// TwinCAT 3 PLC project DiagnosisTools
// Title: TwinCATDiagnosisTools
// Company: Beckhoff Automation K.K.
// Author: Takashi Ichihashi
// ProjectVersion: 1.0.0.1
// ProgramVersion: 3.1.4024.0
// libraries:
//   Tc2_EtherCAT, * (Beckhoff Automation GmbH)
//   Tc2_Standard, * (Beckhoff Automation GmbH)
//   Tc2_System, * (Beckhoff Automation GmbH)
//   Tc2_Utilities, * (Beckhoff Automation GmbH)
//   Tc3_Module, * (Beckhoff Automation GmbH)
// project tree:
//   DUTs/ CoeSdoCommand.TcDUT, sdo_EL6695_diag.TcDUT, sdo_slave_identity.TcDUT, sdo_xplanar_aps_diag.TcDUT
//   GVLs/ ParameterList.TcGVL
//   / PlcTask.TcTTO
//   POUs/ FB_CoeSdoAccess.TcPOU, FB_mqtt_publish.TcPOU, FB_serializer.TcPOU (not stored), ITF_CoeSdoEventHandler.TcIO, queue.TcPOU, MAIN.TcPOU, sdo_watch_time_logging.TcPOU
// real-time tasks:
//   TASK PlcTask: cycle T#10ms, priority 20, ADS port 350
// I/O:
//   DEVICE Device 3 (EtherCAT), AmsNetId 10.200.64.8.4.1
//     Term 1 (EK1100) [EK1100 EtherCAT Coupler (2A E-Bus)]
//       Term 2 (EL2521) [EL2521 1Ch. Pulse Train Output]
//       Term 3 (EL4122) [EL4122 2Ch. Ana. Output  4-20mA, 16bit]
//       Term 4 (EL9576) [EL9576 Brake chopper terminal]
//       Term 5 (EL3152) [EL3152 2Ch. Ana Input 4-20mA]
//       Term 6 (EL2004) [EL2004 4Ch. Dig. Output 24V, 0.5A]
//       Term 7 (EL5101) [EL5101 1Ch. Inc. Encoder 5V]
//       Term 8 (EL6695) [EL6695 EtherCAT Bridge terminal (Primary)]
//       Term 9 (EL9011) [EL9011 End Terminal]

CONFIGURATION DiagnosisTools
    RESOURCE PLC ON TwinCAT3
        TASK PlcTask(INTERVAL := T#10ms, PRIORITY := 20);
        PROGRAM MAIN WITH PlcTask : MAIN;
    END_RESOURCE
END_CONFIGURATION

// ---- DUTs/CoeSdoCommand.TcDUT
(*
SdoRead/WriteRequest
*)
TYPE CoeSdoCommand:
STRUCT
	sNetId				: T_AmsNetId;	// AMS Net ID of EtherCAT Master
	nSlaveAddr			: UINT;			// EtherCAT sub device address
	bCompleteAccess		: BOOL;			// Enable complete access
	nSubIndex			: BYTE;			// Subindex of OD
	nIndex				: WORD;			// Index of OD
	pDstBuf				: PVOID;		// Pointer to data body 
	cbBufLen			: UDINT;		// Size of data body
	datetime			: TIMESTRUCT;	// to be recorded as received date time
	event_handler		: ITF_CoeSdoEventHandler; // Event handler interface
	bError				: BOOL;			// Made true if sdo communication error
	nErrId				: UDINT;		// Set error code if sdo communication error activated
END_STRUCT
END_TYPE

// ---- DUTs/sdo_EL6695_diag.TcDUT
{attribute 'pack_mode' := '2'}
TYPE sdo_EL6695_diag :
STRUCT
	identify : USINT;
	status : UINT;
	cpu_usage : UINT;
	heap_usage : UINT;
	aoe_packets: UINT;
	eoe_packets : UINT;
	foe_packets : UINT;
	soe_packets : UINT;
	voe_packets : UINT;
	other_pacekts: UINT;
	mbx_info : UINT;
	pd_copy_time_my: UINT;
	pd_copy_time_remote :UINT;
	info_2 : UINT;
	info_3 : UINT;
	info_4 : UINT;
	info_5 : UINT;
	info_6 : UINT;
	info_7 : UINT;
	info_8 : UINT;
	info_9 : UINT;
	info_10 : UINT;
	info_11 : UINT;
	info_12 : UINT;
	info_13 : UINT;
	info_14 : UINT;
	info_15 : UINT;
	info_16: UINT;
	info_17 : UINT;
	info_18 : UINT;
END_STRUCT
END_TYPE

// ---- DUTs/sdo_slave_identity.TcDUT
{attribute 'pack_mode' := '2'}
TYPE sdo_slave_identity :
STRUCT
	identify : USINT;
	vendor_id : UDINT;
	product_code : UDINT;
	revision : UDINT;
	serial_number : UDINT;
END_STRUCT
END_TYPE

// ---- DUTs/sdo_xplanar_aps_diag.TcDUT
{attribute 'pack_mode' := '2'}
TYPE sdo_xplanar_aps_diag :
STRUCT
  identity: USINT;
  dc_link_voltage: UDINT;
  power_supply_current: UDINT;
  temperature_north: UINT;
  temperature_east: UINT;
  temperature_south: UINT;
  temperature_west: UINT;
  temperature_center: UINT;
  temperature_power: UINT;
  fan_rpm: UINT;
  fan_duty_cycle: USINT;
  supply_voltage_us: UDINT;
  auxiliary_voltage: UDINT;
  acceleration_x: UDINT;
  acceleration_y: UDINT;
  acceleration_z: UDINT;
  time_to_shutdown: UDINT;
  fb_fw_rev: UDINT;
END_STRUCT
END_TYPE

// ---- GVLs/ParameterList.TcGVL
{attribute 'qualified_only'}
VAR_GLOBAL CONSTANT
	COMMAND_QUEUE_BUFFER_SIZE :UINT := 10;
	MAX_OBSERVATION_SDO :UINT := 100;
END_VAR

// ---- POUs/ITF_CoeSdoEventHandler.TcIO
INTERFACE ITF_CoeSdoEventHandler

METHOD sdo_data_received : BOOL
VAR_INPUT
	command : REFERENCE TO CoeSdoCommand;
END_VAR
END_METHOD

END_INTERFACE

// ---- POUs/MAIN.TcPOU
PROGRAM MAIN
VAR CONSTANT
	EC_MASTER_NETID : T_AmsNetId := '10.200.64.8.4.1';	
END_VAR
VAR

	// COE SDO communication controller object 
	sdo_controller : FB_CoeSdoAccess(sNetId := EC_MASTER_NETID); // EtherCAT Master Object for SDO control


	(* 
		For initialization process( Get all subdevices identity from SDO )
	*)

	bInitialize :BOOL := TRUE;
	s_adr :UINT;

	// define data store.
	sdo_slave_id_data : ARRAY [1002..1008] OF sdo_slave_identity;

	
	
	(*
		 Observation by EL6695 diagnosis data
	*)
	
	// define data store.
	sdo_EL6695_diag_data : sdo_EL6695_diag;
	
	// define event handler when sdo data received by "ITF_CoeSdoEventHandler" implementation.  
	sdo_protocol_with_time_detection: sdo_watch_time_logging;

	// cycle timer for "sdo_EL6695_diag_data" reading.
	read_cycle_timer : TON;
	
	// get ISO 8601 format datetime and cycle time for sdo data received generated by "sdo_protocol_with_time_detection.sdo_data_received()" method.
	datetime_string: STRING(39);
	cycle_time :ULINT;
	
END_VAR

sdo_controller();

// Get Identity data for all sub devices
IF bInitialize THEN
	FOR s_adr := 1002 TO 1008 DO
		sdo_controller.query(
			nSlaveAddr := s_adr,
			bCompleteAccess := TRUE,
			nIndex := 16#1018,
			nSubIndex := 0,
			pDstBuf := ADR(sdo_slave_id_data[s_adr]),
			cbBufLen := SIZEOF(sdo_slave_id_data[s_adr]),
			event_handler := 0
		);
	END_FOR
	bInitialize := FALSE;	
END_IF

// Get diagnostics data every 0.5s
read_cycle_timer(IN := NOT read_cycle_timer.Q, PT := T#500MS);

IF read_cycle_timer.Q THEN
	sdo_controller.query(
				nSlaveAddr := 1008,
				bCompleteAccess := TRUE,
				nIndex := 16#FA20,
				nSubIndex := 0,
				pDstBuf := ADR(sdo_EL6695_diag_data),
				cbBufLen := SIZEOF(sdo_EL6695_diag_data),
				event_handler := sdo_protocol_with_time_detection
			);
END_IF

datetime_string := sdo_protocol_with_time_detection.sDateTime;
cycle_time := sdo_protocol_with_time_detection.lCycleTime;

END_PROGRAM

// ---- POUs/FB_CoeSdoAccess.TcPOU
(*

TwinCAT diagnosis tools library
======================================

quick start
-----------------------


SDO query after boot at once
++++++++++++++++++++++++++++++++++++++++++++++++++++++++++++++++++++++++++++++++


.. code-block:: pascal

	PROGRAM MAIN
	VAR CONSTANT
		EC_MASTER_NETID : T_AmsNetId := '10.200.64.8.4.1';	
	END_VAR
	VAR
		// COE SDO communication controller object 
		sdo_controller : FB_CoeSdoAccess(sNetId := EC_MASTER_NETID); // EtherCAT Master Object for SDO control
	
	
		(* 
			For initialization process( Get all subdevices identity from SDO )
		*)
	
		bInitialize :BOOL := TRUE;
		s_adr :UINT;
	
		// define data store.
		sdo_slave_id_data : ARRAY [1002..1008] OF sdo_slave_identity;
	END_VAR	
	
	sdo_controller();

	// Get Identity data for all sub devices
	IF bInitialize THEN
		FOR s_adr := 1002 TO 1008 DO
			sdo_controller.query(
				nSlaveAddr := s_adr,
				bCompleteAccess := TRUE,
				nIndex := 16#1018,
				nSubIndex := 0,
				pDstBuf := ADR(sdo_slave_id_data[s_adr]),
				cbBufLen := SIZEOF(sdo_slave_id_data[s_adr]),
				event_handler := 0
			);
		END_FOR
		bInitialize := FALSE;	
	END_IF


SDO query cyclically and processing data by original event handler
++++++++++++++++++++++++++++++++++++++++++++++++++++++++++++++++++++++++++++++++


First of all, you can define event handler function block as implementing "ITF_CoeSdoEventHandler" interface which the sdo_data_received method would be executed when sdo data was received.



.. code-block:: pascal

	FUNCTION_BLOCK sdo_watch_time_logging IMPLEMENTS ITF_CoeSdoEventHandler
	VAR_INPUT
	END_VAR
	VAR_OUTPUT
	END_VAR
	VAR
		cycle_time: ULINT;
		datetime_string: STRING;
		last_time :TIMESTRUCT;
	END_VAR

	METHOD sdo_data_received : BOOL
	VAR_INPUT
		command : REFERENCE TO CoeSdoCommand;
	END_VAR
	VAR
	END_VAR
	
	cycle_time := SYSTEMTIME_TO_FILETIME64(command.datetime) - SYSTEMTIME_TO_FILETIME64(last_time);
	datetime_string := SYSTEMTIME_TO_ISO8601(
		systemTime := command.datetime,
		nBias := -540,
		bUTC := TRUE,
		nPrecision := 3
	);
	last_time := command.datetime;


This event handler need to be defined in event handler argument in query method.
	
.. code-block:: pascal

	PROGRAM MAIN
	VAR CONSTANT
		EC_MASTER_NETID : T_AmsNetId := '10.200.64.8.4.1';	
	END_VAR
	VAR
		bInitialize :BOOL := TRUE;
		sdo_controller : FB_CoeSdoAccess(sNetId := EC_MASTER_NETID); // EtherCAT Master Object for SDO control

		(*
			 Observation by EL6695 diagnosis data
		*)
		
		// define data store.
		sdo_EL6695_diag_data : sdo_EL6695_diag;
		
		// define event handler when sdo data received by "ITF_CoeSdoEventHandler" implementation.  
		sdo_protocol_with_time_detection: sdo_watch_time_logging;
	
		// cycle timer for "sdo_EL6695_diag_data" reading.
		read_cycle_timer : TON;
		
		// get ISO 8601 format datetime and cycle time for sdo data received generated by "sdo_protocol_with_time_detection.sdo_data_received()" method.
		datetime_string: STRING(39);
		cycle_time :ULINT;

	END_VAR
	
	// Get diagnostics data every 0.5s
	read_cycle_timer(IN := NOT read_cycle_timer.Q, PT := T#500MS);
	
	IF read_cycle_timer.Q THEN
		sdo_controller.query(
					nSlaveAddr := 1008,
					bCompleteAccess := TRUE,
					nIndex := 16#FA20,
					nSubIndex := 0,
					pDstBuf := ADR(sdo_EL6695_diag_data),
					cbBufLen := SIZEOF(sdo_EL6695_diag_data),
					event_handler := sdo_protocol_with_time_detection
				);
	END_IF
	
	datetime_string := sdo_protocol_with_time_detection.sDateTime;
	cycle_time := sdo_protocol_with_time_detection.lCycleTime;
	
*)
FUNCTION_BLOCK FB_CoeSdoAccess
VAR_INPUT
END_VAR
VAR_OUTPUT
END_VAR
VAR
	_event_handler : ITF_CoeSdoEventHandler;
	bInitialize : BOOL := TRUE;
	_queue: queue;
	fbSdoRead : FB_ECCoeSdoReadEx;
	sdo_command: REFERENCE TO CoeSdoCommand;
	_step :UINT;
	_sNetId: T_AmsNetId;
	
	  // Get UTC time
 	fbLocalTime: FB_LocalSystemTime := (bEnable:=TRUE, dwCycle:=5);     // For getting current time as local time
  	fbGetTimeZoneInformation: FB_GetTimeZoneInformation := (bExecute := TRUE);      // For getting local timezone information
  	fbTzSpecificLocalTimeToSystemTime: FB_TzSpecificLocalTimeToSystemTime;          // FOr converting local time to UTC.
	bExecuting :BOOL;
END_VAR

// Get and sync local time with PC OS.
fbLocalTime();
IF bInitialize THEN
	fbGetTimeZoneInformation(bExecute := TRUE);
	IF NOT fbGetTimeZoneInformation.bBusy THEN
		fbGetTimeZoneInformation(bExecute := FALSE);
		bInitialize := FALSE;
	END_IF
END_IF


CASE _step OF
	0:
		IF _queue.queue_usage > 0 AND NOT fbSdoRead.bBusy THEN
			sdo_command REF= _queue.get();
			_step := 1;
		END_IF
	1:
		fbSdoRead(
			sNetId := sdo_command.sNetId, // Change it as an individual situation
		 	nSlaveAddr := sdo_command.nSlaveAddr, // Change it as an individual situation
		  	nIndex := sdo_command.nIndex,
		  	nSubIndex := sdo_command.nSubIndex,
		  	pDstBuf := sdo_command.pDstBuf,
		  	cbBufLen := sdo_command.cbBufLen,
		  	bExecute := TRUE,
		  	bCompleteAccess := sdo_command.bCompleteAccess,
		  	bError => sdo_command.bError,
		  	nErrId => sdo_command.nErrId
		);
		IF fbSdoRead.bBusy THEN
			_step := 2;
		END_IF
	2:	
		fbSdoRead(bExecute := FALSE);
		IF NOT fbSdoRead.bBusy THEN
			IF NOT fbSdoRead.bError THEN
				fbTzSpecificLocalTimeToSystemTime(in := fbLocalTime.systemTime, tzInfo := fbGetTimeZoneInformation.tzInfo);
				sdo_command.datetime := fbTzSpecificLocalTimeToSystemTime.out;
				IF sdo_command.event_handler <> 0 THEN
					sdo_command.event_handler.sdo_data_received(sdo_command);				
				END_IF
			END_IF
			_step := 0;
		END_IF
END_CASE

METHOD FB_init : BOOL
VAR_INPUT
	bInitRetains : BOOL; // if TRUE, the retain variables are initialized (warm start / cold start)
	bInCopyCode : BOOL;  // if TRUE, the instance afterwards gets moved into the copy code (online change)
	sNetId				: T_AmsNetId;	// AMS Net ID of EtherCAT Master
END_VAR
_sNetId := sNetId;
END_METHOD

PROPERTY NetId : T_AmsNetId
GET
NetId := _sNetId;
END_GET
SET
_sNetId := NetId;
END_SET
END_PROPERTY

METHOD query : POINTER TO CoeSdoCommand
VAR_INPUT
	nSlaveAddr	: UINT;
	(* Enable complete access*)
	bCompleteAccess	: BOOL := TRUE;
	(* Index of OD*)
	nIndex	: WORD;
	(* Subindex of OD*)
	nSubIndex	: BYTE := 0;
	(* Pointer to data body *)
	pDstBuf	: PVOID;
	(* Size of data body*)
	cbBufLen	: UDINT;
	(* Event Handler Interface *)
	event_handler : ITF_CoeSdoEventHandler := 0;
END_VAR

VAR_STAT
	command: CoeSdoCommand;	
END_VAR
IF NOT _queue.full THEN
	command.sNetId := _sNetId;
	command.nSlaveAddr := nSlaveAddr;
	command.bCompleteAccess := bCompleteAccess;
	command.nIndex := nIndex;
	command.nSubIndex := nSubIndex;
	command.pDstBuf := pDstBuf;
	command.cbBufLen := cbBufLen;
	command.event_handler := event_handler;
	query := _queue.put(command);
END_IF
END_METHOD

// ---- POUs/sdo_watch_time_logging.TcPOU
FUNCTION_BLOCK sdo_watch_time_logging IMPLEMENTS ITF_CoeSdoEventHandler
VAR_INPUT
END_VAR
VAR_OUTPUT
END_VAR
VAR
	cycle_time: ULINT;
	datetime_string: STRING;
	last_time :TIMESTRUCT;

END_VAR

PROPERTY lCycleTime : ULINT
GET
lCycleTime := cycle_time;
END_GET
END_PROPERTY

PROPERTY sDateTime : STRING
GET
sDateTime := datetime_string;
END_GET
END_PROPERTY

METHOD sdo_data_received : BOOL
VAR_INPUT
	command : REFERENCE TO CoeSdoCommand;
END_VAR
VAR
END_VAR

cycle_time := SYSTEMTIME_TO_FILETIME64(command.datetime) - SYSTEMTIME_TO_FILETIME64(last_time);
datetime_string := SYSTEMTIME_TO_ISO8601(
	systemTime := command.datetime,
	nBias := -540,
	bUTC := TRUE,
	nPrecision := 3
);
last_time := command.datetime;
END_METHOD

END_FUNCTION_BLOCK

// ---- POUs/queue.TcPOU
(*
:Author: Takashi Ichihashi
:Date: 2023-03-07

Decreration
=========================

.. code-block:: 

	// Variables for queue feature
	fb_deq : dequeue;
	get_data : T_Arg;
	// databuffer for 1 second with 10 ms time delta
    queue_buffer: ARRAY[0..99] OF T_Arg;
	

Useage
=================

This is example code that the sInputData is queued in and queued out for sOutputData.

.. code-block:: 

	// put_data
	IF NOT fb_deq.full THEN

		sInputData := ANY_DATA;
		// put pointer
		fb_deq.put(F_BIGTYPE(ADR(sInputData),SIZEOF(sInputData)));

	END_IF
	
	// getting data
	get_data := fb_deq.get();
	MEMCPY(ADR(sOutputData), get_data.pData, get_data.cbLen);
	
	
*)

FUNCTION_BLOCK queue
VAR
	_queue_usage:	UDINT;
	_queue_size:	UDINT := ParameterList.COMMAND_QUEUE_BUFFER_SIZE;
	nWriteIndex: 	UDINT;
	nReadIndex: 	UDINT;
	queue_buffer:	ARRAY [0..ParameterList.COMMAND_QUEUE_BUFFER_SIZE - 1] OF CoeSdoCommand;
END_VAR

PROPERTY full : BOOL
GET
full :=  _queue_usage >= ParameterList.COMMAND_QUEUE_BUFFER_SIZE - 1;
END_GET
END_PROPERTY

METHOD get : REFERENCE TO CoeSdoCommand
VAR_INPUT
END_VAR
//Set buffer index

IF _queue_usage > 0 THEN
	get REF= queue_buffer[nReadIndex];
	_queue_usage := _queue_usage - 1;
	nReadIndex := nReadIndex + 1;
	IF nReadIndex > ParameterList.COMMAND_QUEUE_BUFFER_SIZE - 1 THEN
		nReadIndex := 0;
	END_IF
END_IF

RETURN;
END_METHOD

PROPERTY PUBLIC index : UDINT
GET
index := nWriteIndex;
END_GET
END_PROPERTY

PROPERTY PUBLIC max_index : UDINT
GET
max_index := ParameterList.COMMAND_QUEUE_BUFFER_SIZE - 1;
END_GET
END_PROPERTY

METHOD PUBLIC put : POINTER TO CoeSdoCommand
VAR_INPUT
	lData:	CoeSdoCommand;
END_VAR
//Set buffer index
put := 0;
IF _queue_usage < ParameterList.COMMAND_QUEUE_BUFFER_SIZE - 1 THEN
	queue_buffer[nWriteIndex] := lData;
	put := ADR(queue_buffer[nWriteIndex]);
	_queue_usage := _queue_usage + 1;
	nWriteIndex := nWriteIndex + 1;
	IF nWriteIndex > ParameterList.COMMAND_QUEUE_BUFFER_SIZE - 1 THEN
		nWriteIndex := 0;
	END_IF
END_IF

RETURN;
END_METHOD

PROPERTY queue_size : UDINT
GET
queue_size := _queue_size;
END_GET
END_PROPERTY

PROPERTY queue_usage : UDINT
GET
queue_usage := _queue_usage;
END_GET
END_PROPERTY

END_FUNCTION_BLOCK

// ---- POUs/FB_mqtt_publish.TcPOU
FUNCTION_BLOCK FB_mqtt_publish IMPLEMENTS  ITF_CoeSdoEventHandler
VAR_INPUT
END_VAR
VAR_OUTPUT
END_VAR
VAR
	// published message
	fbMqttClient : FB_IotMqttClient;
	fbMessageQueue : FB_IotMqttMessageQueue;
	bSetParameter : BOOL := TRUE;
	bConnect : BOOL := TRUE;
	hrErrorOccurred : HRESULT; // contains the latest occurred error
	
	fbSerializer :FB_Serializer;
	
	sTopicPub : STRING(255) := 'devices/1';
	sPayloadPub : STRING(255);
	
	// for making publish event
	publish_cycle_timer :TON;
	datetime_string: STRING(39);
	
END_VAR

{warning 'add method implementation '}
METHOD sdo_data_received : BOOL
VAR_INPUT
	command	: REFERENCE TO CoeSdoCommand;
END_VAR
VAR
	diag_data_body: POINTER TO sdo_xplanar_aps_diag;
	tile_number : UINT;
END_VAR


// Connect MQTT broker and publish

IF bSetParameter THEN
	bSetParameter := FALSE;
	//fbMqttClient.stTLS.sCA := 'c:\TwinCAT\3.1\Config\Certificates\BaltimoreCyberTrust.crt'; // CA certificate 
	fbMqttClient.stTLS.sAzureSas := 'HostName=IndustrialOPNFair2024-IoTHub.azure-devices.net;DeviceId=unit230;SharedAccessSignature=SharedAccessSignature sr=IndustrialOPNFair2024-IoTHub.azure-devices.net%2Fdevices%2Funit230&sig=GxT9x70t1Q1per9XXu4Az%2FJhK1jBZt14KJ%2B7LG4NB%2Fw%3D&se=1712921181'; // Device SAS Token
	fbMqttClient.ipMessageQueue := fbMessageQueue;
END_IF

fbMqttClient.Execute(bConnect);
IF fbMqttClient.bError THEN
  // add your error logging here
  hrErrorOccurred := fbMqttClient.hrErrorCode;
END_IF


publish_cycle_timer(IN := NOT publish_cycle_timer.Q, PT := T#10S);
diag_data_body := command.pDstBuf;

CASE command.nSlaveAddr OF
	1001:
		tile_number := 1;
	1003:
		tile_number := 2;
END_CASE

IF fbMqttClient.bConnected THEN
	datetime_string := SYSTEMTIME_TO_ISO8601(
		systemTime := command.datetime,
		nBias := 0,
		bUTC := TRUE,
		nPrecision := 3
	);
	
	sPayloadPub := fbSerializer.serialize(
	  datetime := datetime_string,
	  device_name := CONCAT('xplanar_tile_', UINT_TO_STRING(command.nSlaveAddr)),
	  diag_data_body := diag_data_body
	);
	fbMqttClient.Publish(	sTopic:= sTopicPub, 
				pPayload:= ADR(sPayloadPub), nPayloadSize:= LEN2(ADR(sPayloadPub)), 
				eQoS:= TcIotMqttQos.AtMostOnceDelivery, bRetain:= FALSE, bQueue:= FALSE );
    IF fbMqttClient.bError THEN
      // add your error logging here
      hrErrorOccurred := fbMqttClient.hrErrorCode;
    END_IF
END_IF
END_METHOD

END_FUNCTION_BLOCK
